PROGRAM SimulationViewBindings
VAR
	// Pointers to simulated variables
	pFlowMeasurement : POINTER TO REAL := ADR(SerialCommunicationController.HandleSerialCommunication.readData.flowMeasurement);
	pPressureMeasurement : POINTER TO DINT := ADR(GVL_IO.reactorPressure); 	
	
	// Locals
	flowSlider_Variable : REAL;
	pressureSlider_Variable : DINT;
END_VAR


pFlowMeasurement^ := flowSlider_Variable/100;
pPressureMeasurement^ := pressureSlider_Variable;

END_PROGRAM

(* stored: Version 1.1.0.1, ProductVersion 3.1.4024.9
   POU SimulationViewBindings: Id {b55f8d2e-1783-4f6e-a2c7-a2b84d2145a7}, SpecialFunc None *)
